SUBROUTINE_BLOCK ValveA_Diag:SBR16
TITLE=// ============================================================
// // 文件: FC30_ValveA_Diag.stl
// // 功能: 阀A诊断（差值法计量+延时验证4项并行+漫溢保护）
// // Story: AQEX-7 阀门诊断
// // 调用方: FC11(S1上缸进水)
// // 说明: 阀A不使用四态诊断，采用差值法+延时验证
// //       诊断子状态VW260: 0空闲/1等开到位/2开启完成/3运行中/5关闭后验证
// //
// // 修复记录:
// //   P1 - MOVR/-R 替换 MOVD/-D: 流量计数据为REAL浮点,之前用双整数指令导致VD90=NAN
// //   P2 - 单NETWORK合并: 所有JMP/LBL在同一NETWORK内,解决STEP7导入跨NETWORK跳转失效
// //   P3 - I8.0 去掉EU: 子状态1→2改用常开触点,PLC冷启动时阀已开到位也能正常进入子状态2
// //   P4 - 关阀快照MOVD改MOVR: 语义一致,REAL数据用MOVR搬运
// // ============================================================
// 
// // 符号说明:
// // VW260 : Diag_State_A     阀A诊断子状态
// // VW266 : Diag_Result_A    阀A诊断结果(0进行中/1正常/2故障)
// // VD308 : VD_FlowMeter_CloseSnapshot  阀A关阀瞬间流量计快照
// // VD312 : VD_FlowMeter_CloseDelta     阀A关阀后流量计差值
// // VD316 : 目标进水量(HMI设定)
// // T50   : 阀A开到位超时(100ms时基)
// // T51   : 阀A关阀后延时验证(100ms时基)
// // T52   : 开到位但无流2s确认(100ms时基)
// // I0.0  : 流量开关A(有流=ON)
// // I0.5  : 液位计A高位(漫溢=ON)
// // I8.0  : 阀A开到位反馈
// // I8.1  : 阀A关到位反馈
// // Q0.2  : 阀A(电动球阀)
// // Q0.5  : NC球阀-上缸
BEGIN
Network 1
//  ============================================================
//  NETWORK 1 - 单NETWORK版 FC30
//  所有JMP/LBL在同一NETWORK内,避免STEP7导入后跳转失效
//  ============================================================
//  ========== 第一部分: 漫溢保护(优先级最高,全程监控) ==========
LD     CPU_输入5:I0.5          // 液位计A高位=漫溢
S      V300.0, 1             // M_Alarm_Overflow_AHigh
S      V300.2, 1             // M_Alarm_NCValve_Top
R      CPU_输出5:Q0.5, 1       // 关NC球阀(切断水流)
R      CPU_输出2:Q0.2, 1       // 关阀A
MOVW   99, VW2               // 转S_ERROR
MOVB   2, VB266              // Diag_Result_A=2故障
JMP    1                     // 跳到结束
// ========== 第二部分: 子状态调度(根据VB260分发) ========== // ========== 第二部分: 子状态调度(根据VB260分发) ==========
// ★关键修复: 子状态只存在VB260中,FC11用MOVB写VB260,VB261=0 // ★关键修复: 子状态只存在VB260中,FC11用MOVB写VB260,VB261=0
//   因此VW260实际=VB260×256(如VB260=2则VW260=512),必须用LDB=字节比较 //   因此VW260实际=VB260×256(如VB260=2则VW260=512),必须用LDB=字节比较
LDB=   VB260, 0
LDB=   VB260, 0              // 子状态0: 空闲
LDB=   VB260, 1
JMP    2                     // 子状态1: 等开到位
LDB=   VB260, 2
LDB=   VB260, 1              // 子状态2: 等流量开关
LDB=   VB260, 3
JMP    3                     // 子状态3: ★运行中算VD90★
LDB=   VB260, 5
LDB=   VB260, 2              // 子状态5: 关阀后延时验证
JMP    4                     // 兜底: 非法状态跳到结束
// ========== 第三部分: 子状态0 - 空闲 ========== // ========== 第三部分: 子状态0 - 空闲 ==========
LBL    2
// 等待FC11触发置VW260=1, 无额外动作   // 等待FC11触发置VW260=1, 无额外动作
JMP    1
// ========== 第四部分: 子状态1 - 等待开到位 ========== // ========== 第四部分: 子状态1 - 等待开到位 ==========
LBL    3
// T50超时计时(PT=VW278, 由FC11计算VD358×10写入) // T50超时计时(PT=VW278, 由FC11计算VD358×10写入)
LD     SM0.0
TON    T50, VW278
// I8.0开到位反馈=ON → 转子状态2      // I8.0开到位反馈=ON → 转子状态2
// ★P3修复: 去掉EU(上升沿),改用常开触点   // ★P3修复: 去掉EU(上升沿),改用常开触点
//   正常: 阀A打开后I8.0从OFF→ON,直接触发 //   正常: 阀A打开后I8.0从OFF→ON,直接触发
//   异常: PLC冷启动时阀已开到位(I8.0本来就是ON),也能立即进入子状态2 //   异常: PLC冷启动时阀已开到位(I8.0本来就是ON),也能立即进入子状态2
LD     I8.0
LDB=   VB260, 3              // VW260=2
JMP    5                     // 清子状态索引
LDB=   VB260, 5              // 复位超时计时
JMP    1
// T50超时 → 开到位超时报警           // T50超时 → 开到位超时报警
LD     T50
JMP    6                     // M_Alarm_ValveA_OpenTimeout
MOVW   99, VW2
MOVB   2, VB266
JMP    1
// ========== 第五部分: 子状态2 - 等待流量开关 ========== // ========== 第五部分: 子状态2 - 等待流量开关 ==========
LBL    4
// I0.0流量开关A=ON → 正常有流, 转子状态3运行中 // I0.0流量开关A=ON → 正常有流, 转子状态3运行中
LD     I0.0
JMP    1                     // VW260=3运行中
MOVB   0, VB261
JMP    1
// 开到位但无流 → 加2s延时确认避免瞬时波动    // 开到位但无流 → 加2s延时确认避免瞬时波动
LBL    2                     // 阀确实已开到位
JMP    1                     // 但无流量
LBL    3                     // 2s确认(20×100ms)
LD     T52
LD     Always_On:SM0.0       // M_Alarm_ValveA_OpenNoFlow
MOVW   99, VW2
MOVB   2, VB266
JMP    1
// ========== 第六部分: 子状态3 - ★运行中差值法持续计量★ ========== // ========== 第六部分: 子状态3 - ★运行中差值法持续计量★ ==========
LBL    5
// ★P1修复: 用MOVR/-R实数指令计算进水量(原MOVD/-D导致NAN) // ★P1修复: 用MOVR/-R实数指令计算进水量(原MOVD/-D导致NAN)
// VD_Current_InletVolume(VD90) = VD86(当前累计) - VD82(开启快照) // VD_Current_InletVolume(VD90) = VD86(当前累计) - VD82(开启快照)
LD     SM0.0
TON    T50, VW278            // ★MOVR: 实数搬运
LD     EM0_输入0:I8.0          // ★-R: 实数减法
MOVB   2, VB260              // 当前进水量
// 进水量达标 → 关阀A + 快照关阀瞬间流量计值 + 转子状态5 // 进水量达标 → 关阀A + 快照关阀瞬间流量计值 + 转子状态5
LD     SM0.0
LPS
MOVB   0, VB261              // 当前进水量 ≥ 目标进水量
R      T50, 1                // 关阀A
// ★P4修复: 关阀快照也用MOVR(原MOVD虽能跑但语义不一致) // ★P4修复: 关阀快照也用MOVR(原MOVD虽能跑但语义不一致)
JMP    1                     // VD_FlowMeter_CloseSnapshot
LD     T50                   // VW260=5(关闭后验证)
MOVB   0, VB261
S      V301.4, 1             // 复位开到位无流确认计时
LPP
JMP    1
// ========== 第七部分: 子状态5 - 关阀后延时验证(4项并行) ========== // ========== 第七部分: 子状态5 - 关阀后延时验证(4项并行) ==========
LBL    6
// T51延时验证计时(PT=VW280, 由FC11计算VD66×10写入) // T51延时验证计时(PT=VW280, 由FC11计算VD66×10写入)
LD     SM0.0
TON    T51, VW280
// ★P1修复: 关阀后内漏检测也用MOVR/-R实数指令 // ★P1修复: 关阀后内漏检测也用MOVR/-R实数指令
// 持续计算关阀后流量计差值 = VD86(当前) - VD308(关阀快照) // 持续计算关阀后流量计差值 = VD86(当前) - VD308(关阀快照)
LD     SM0.0
MOVR   VD86, AC0
-R     VD308, AC0
MOVW   99, VW2               // VD_FlowMeter_CloseDelta
// --- 延时到达后4项并行校验 ---       // --- 延时到达后4项并行校验 ---
MOVB   2, VB266              // 仅T51到达时执行
LPS
// 校验1: 关阀后仍有流(流量开关A=ON)     // 校验1: 关阀后仍有流(流量开关A=ON)
A      I0.0
JMP    1                     // M_Alarm_ValveA_CloseFlow
// 校验2: 内漏(流量计差值>0.1L, 说明仍在缓慢注水) // 校验2: 内漏(流量计差值>0.1L, 说明仍在缓慢注水)
LPS
LBL    4                     // 阈值0.1L=100ml, 现场整定
LD     CPU_输入0:I0.0          // M_Alarm_ValveA_Leak
LPP
// 校验3: 关到位反馈超时(I8.1=OFF)    // 校验3: 关到位反馈超时(I8.1=OFF)
AN     I8.1
MOVB   3, VB260              // M_Alarm_ValveA_CloseTimeout
// 校验4: 关到位但仍有流(交叉验证)        // 校验4: 关到位但仍有流(交叉验证)
MOVB   0, VB261              // 阀确实关到位
JMP    1                     // 但流量开关仍有流
LD     EM0_输入0:I8.0          // M_Alarm_ValveA_CloseLeak
LPP
// --- 校验结果判定 ---            // --- 校验结果判定 ---
AN     CPU_输入0:I0.0          // T51已到
LPS
// 4项全通过: 流量开关OFF AND 差值不增 AND 关到位ON // 4项全通过: 流量开关OFF AND 差值不增 AND 关到位ON
TON    T52, 20               // 流量开关A=OFF
LD     T52                   // 差值≤0.1L(不增长=无内漏)
S      V301.5, 1             // 关到位=ON
// → 诊断正常完成                  // → 诊断正常完成
MOVW   99, VW2               // VW260=0空闲(等待下轮)
MOVB   0, VB261
MOVB   2, VB266              // Diag_Result_A=1正常完成
JMP    1                     // 复位延时计时
JMP    1
LPP
// 任一项报警 → 转S_ERROR          // 任一项报警 → 转S_ERROR
LD     T51
LBL    5                     // 4个报警标志任一为1
O      V301.1
O      V301.2
O      V301.3
LD     Always_On:SM0.0       // 转S_ERROR
MOVR   VD86, AC0             // 故障
JMP    1
// ========== 结束 ==========  // ========== 结束 ==========
LBL    1
// ============================================================ // ============================================================
// 文件结束                      // 文件结束
// 说明:                       // 说明:
//   1. FC11调用本FC前需置VW260=1启动诊断 //   1. FC11调用本FC前需置VW260=1启动诊断
//   2. FC11检查VW266: 0=进行中等待, 1=正常完成转S2, 2=故障(已转S_ERROR) //   2. FC11检查VW266: 0=进行中等待, 1=正常完成转S2, 2=故障(已转S_ERROR)
//   3. VD316(目标进水量)由HMI设定或FC11计算写入 //   3. VD316(目标进水量)由HMI设定或FC11计算写入
//   4. VW278=T50×10(开到位超时), VW280=T51×10(延时验证), 由FC11计算写入 //   4. VW278=T50×10(开到位超时), VW280=T51×10(延时验证), 由FC11计算写入
//   5. 内漏阈值0.1L为初值, 需现场整定   //   5. 内漏阈值0.1L为初值, 需现场整定
//   6. 所有JMP/LBL在单NETWORK内, 避免STEP7导入后跳转失效(P2修复) //   6. 所有JMP/LBL在单NETWORK内, 避免STEP7导入后跳转失效(P2修复)
// ============================================================

 // ============================================================
-R     VD82, AC0
MOVR   AC0, VD90
LD     Always_On:SM0.0
LPS
AR>=   VD90, VD316
R      CPU_输出2:Q0.2, 1
MOVR   VD86, VD308
MOVB   5, VB260
MOVB   0, VB261
R      T52, 1
LPP
JMP    1
LBL    6
LD     Always_On:SM0.0
TON    T51, VW280
LD     Always_On:SM0.0
MOVR   VD86, AC0
-R     VD308, AC0
MOVR   AC0, VD312
LD     T51
LPS
A      CPU_输入0:I0.0
S      V301.0, 1
LPS
AR>    VD312, 0.1
S      V301.1, 1
LPP
AN     EM0_输入1:I8.1
S      V301.2, 1
A      EM0_输入1:I8.1
A      CPU_输入0:I0.0
S      V301.3, 1
LPP
LD     T51
LPS
AN     CPU_输入0:I0.0
AR<=   VD312, 0.1
A      EM0_输入1:I8.1
MOVB   0, VB260
MOVB   0, VB261
MOVB   1, VB266
R      T51, 1
JMP    1
LPP
LD     T51
A      V301.0
O      V301.1
O      V301.2
O      V301.3
MOVW   99, VW2
MOVB   2, VB266
JMP    1
LBL    1
END_SUBROUTINE_BLOCK

SUBROUTINE_BLOCK ValveB_Diag:SBR17
TITLE=// ============================================================
// // 文件: FC31_ValveB_Diag.stl
// // 功能: 阀B诊断（四态诊断+开关到位+超时保护+漫溢保护）
// // Story: AQEX-7 阀门诊断
// // 调用方: FC15(S4上→下转移)
// // 说明: 阀B四态诊断(流量开关B+液位计A低位)
// //       诊断子状态VW262: 0空闲/1等开到位/2开启完成/3运行中/4等关到位
// // ============================================================
// 
// // 符号说明:
// // VW262 : Diag_State_B     阀B诊断子状态
// // VW268 : Diag_Result_B    阀B诊断结果(0/1/2)
// // T53   : 阀B开到位超时
// // T54   : 阀B流量开关超时保护
// // T55   : 阀B关到位超时
// // I0.1  : 流量开关B
// // I0.6  : 液位计A低位(上缸排空)
// // I0.7  : 液位计B高位(下缸漫溢)
// // I8.2  : 阀B开到位反馈
// // I8.3  : 阀B关到位反馈
// // Q0.3  : 阀B
// // Q0.6  : NC球阀-下缸
// 
BEGIN
Network 1
//  漫溢保护（全程，优先级最高）
//  液位计B高位=ON立即报警+关NC阀+关阀B+转S_ERROR
//  NC球阀与电动球阀串联冗余:高位时关闭NC球阀切断水流,防止球阀关不严持续注水
LD     CPU_输入7:I0.7
S      V300.1, 1             // M_Alarm_Overflow_BHigh
S      V300.3, 1             // M_Alarm_NCValve_Bottom(NC球阀下缸关闭报警,漫溢风险级)
R      CPU_输出6:Q0.6, 1       // 关闭下缸NC球阀(切断水流)
R      CPU_输出3:Q0.3, 1       // 关阀B
MOVW   99, VW2
MOVB   2, VB268              // 故障
JMP    1




Network 2
//  诊断子状态调度
LDW=   VW262, 0
JMP    2
LDW=   VW262, 1
JMP    3
LDW=   VW262, 2
JMP    4
LDW=   VW262, 3
JMP    5
LDW=   VW262, 4
JMP    6
JMP    1




// ---- 子状态0: 空闲 ----
       // ---- 子状态0: 空闲 ----
Network 3
//  S0空闲
LBL    2
JMP    1




// ---- 子状态1: 等待开到位 ----
    // ---- 子状态1: 等待开到位 ----
Network 4
//  S1等待开到位
LBL    3
// T53开到位超时 + T54流量开关超时(两套独立判据)
 // T53开到位超时 + T54流量开关超时(两套独立判据)
LD     Always_On:SM0.0
TON    T53, VW274            // PT=VD_Timeout_ValveB(VD362)×10
TON    T54, VW274            // 流量开关超时(同参数，独立计时)


// 开到位=ON → 转S2
             // 开到位=ON → 转S2
LD     EM0_输入2:I8.2
EU
MOVB   2, VB262
MOVB   0, VB263
R      T53, 1
R      T54, 1
JMP    1


// 开到位超时 → 报警
               // 开到位超时 → 报警
LD     T53
S      V302.1, 1             // M_Alarm_ValveB_OpenTimeout
MOVW   99, VW2
MOVB   2, VB268
JMP    1


// 流量开关超时(开阀后一直无流) → 报警
     // 流量开关超时(开阀后一直无流) → 报警
LD     T54
AN     CPU_输入1:I0.1          // 确认流量开关B仍OFF
S      V302.2, 1             // M_Alarm_ValveB_OpenNoFlow
MOVW   99, VW2
MOVB   2, VB268
JMP    1




// ---- 子状态2: 开启完成检查 ----
   // ---- 子状态2: 开启完成检查 ----
Network 5
//  S2开启完成检查
LBL    4
// 流量开关B=ON → 正常，转S3
        // 流量开关B=ON → 正常，转S3
LD     CPU_输入1:I0.1
MOVB   3, VB262
MOVB   0, VB263
JMP    1


// 开到位但无流 → 报警
              // 开到位但无流 → 报警
LD     EM0_输入2:I8.2
AN     CPU_输入1:I0.1
S      V302.2, 1             // M_Alarm_ValveB_OpenNoFlow
MOVW   99, VW2
MOVB   2, VB268
JMP    1




// ---- 子状态3: 运行中(四态诊断持续扫描) ----
 // ---- 子状态3: 运行中(四态诊断持续扫描) ----
Network 6
//  S3四态诊断
LBL    5
// 四态诊断: 流量开关B(I0.1) + 液位计A低位(I0.6)
 // 四态诊断: 流量开关B(I0.1) + 液位计A低位(I0.6)
// 状态3: 流量开关OFF + 液位低位ON → 上缸排空，关阀触发
 // 状态3: 流量开关OFF + 液位低位ON → 上缸排空，关阀触发
LD     CPU_输入6:I0.6          // 液位计A低位=ON(上缸空)
AN     CPU_输入1:I0.1          // 且流量开关B=OFF(转移结束)
R      CPU_输出3:Q0.3, 1       // 关阀B
MOVB   4, VB262              // 转S4等关到位
MOVB   0, VB263
JMP    1


// 状态4: 流量开关OFF + 液位低位OFF → 设备故障
 // 状态4: 流量开关OFF + 液位低位OFF → 设备故障
LD     CPU_输入1:I0.1          // 流量开关B
NOT
AN     CPU_输入6:I0.6          // 且液位低位OFF
// 注:需排除刚开始转移时的瞬时(流量开关尚未ON)
 // 注:需排除刚开始转移时的瞬时(流量开关尚未ON)
// 简化: 直接判定状态4
              // 简化: 直接判定状态4
S      V302.0, 1             // M_Alarm_ValveB_Diag
MOVW   99, VW2
MOVB   2, VB268
JMP    1


// 状态1/2: 流量开关ON → 正常转移中/即将排空，继续
 // 状态1/2: 流量开关ON → 正常转移中/即将排空，继续
LD     CPU_输入1:I0.1
JMP    1




// ---- 子状态4: 等待关到位 ----
    // ---- 子状态4: 等待关到位 ----
Network 7
//  S4等待关到位
LBL    6
// T55关到位超时
                 // T55关到位超时
LD     Always_On:SM0.0
TON    T55, VW274            // PT=VD_Timeout_ValveB×10


// 关到位=ON AND 流量开关=OFF → 正常完成
 // 关到位=ON AND 流量开关=OFF → 正常完成
LD     EM0_输入3:I8.3
AN     CPU_输入1:I0.1
MOVB   0, VB262              // VW262=0空闲
MOVB   0, VB263
MOVB   1, VB268              // Diag_Result_B=1正常完成
R      T55, 1
JMP    1


// 关到位=ON AND 流量开关=ON → 内漏
  // 关到位=ON AND 流量开关=ON → 内漏
LD     EM0_输入3:I8.3
A      CPU_输入1:I0.1
S      V302.4, 1             // M_Alarm_ValveB_CloseLeak
MOVW   99, VW2
MOVB   2, VB268
JMP    1


// 关到位超时 → 报警
               // 关到位超时 → 报警
LD     T55
AN     EM0_输入3:I8.3
S      V302.3, 1             // M_Alarm_ValveB_CloseTimeout
MOVW   99, VW2
MOVB   2, VB268
JMP    1




Network 8
//  诊断结束
LBL    1




// ============================================================
 // ============================================================
// 文件结束
                     // 文件结束
// 说明:
                      // 说明:
//   1. FC15调用本FC前置VW262=1启动
 //   1. FC15调用本FC前置VW262=1启动
//   2. FC15检查VW268: 0等待, 1正常完成转S5, 2故障
 //   2. FC15检查VW268: 0等待, 1正常完成转S5, 2故障
//   3. VW274=VD_Timeout_ValveB(VD362)×10转换值
 //   3. VW274=VD_Timeout_ValveB(VD362)×10转换值
//   4. 四态诊断状态4需排除转移初期瞬时，实际需加延时确认
 //   4. 四态诊断状态4需排除转移初期瞬时，实际需加延时确认
// ============================================================
 // ============================================================


END_SUBROUTINE_BLOCK

SUBROUTINE_BLOCK ValveC_Diag:SBR18
TITLE=// ============================================================
// // 文件: FC32_ValveC_Diag.stl
// // 功能: 阀C诊断（四态诊断+开关到位+超时保护）
// // Story: AQEX-7 阀门诊断
// // 调用方: FC17(S6下缸排水)
// // 说明: 阀C四态诊断(流量开关C+液位计B低位)，与阀B对称
// //       阀C无漫溢保护(下缸排水不会漫溢)
// //       诊断子状态VW264: 0空闲/1等开到位/2开启完成/3运行中/4等关到位
// // ============================================================
// 
// // 符号说明:
// // VW264 : Diag_State_C     阀C诊断子状态
// // VW270 : Diag_Result_C    阀C诊断结果(0/1/2)
// // T56   : 阀C开到位超时
// // T57   : 阀C流量开关超时保护
// // T58   : 阀C关到位超时
// // I0.2  : 流量开关C
// // I1.0  : 液位计B低位(下缸排空)
// // I8.4  : 阀C开到位反馈
// // I8.5  : 阀C关到位反馈
// // Q0.4  : 阀C
BEGIN
Network 1
//  诊断子状态调度
//  注: 阀C无漫溢保护，直接进入状态调度
LDW=   VW264, 0
JMP    1
LDW=   VW264, 1
JMP    2
LDW=   VW264, 2
JMP    3
LDW=   VW264, 3
JMP    4
LDW=   VW264, 4
JMP    5
JMP    6




// ---- 子状态0: 空闲 ----
       // ---- 子状态0: 空闲 ----
Network 2
//  S0空闲
LBL    1
JMP    6




// ---- 子状态1: 等待开到位 ----
    // ---- 子状态1: 等待开到位 ----
Network 3
//  S1等待开到位
LBL    2
// T56开到位超时 + T57流量开关超时(两套独立判据)
 // T56开到位超时 + T57流量开关超时(两套独立判据)
LD     Always_On:SM0.0
TON    T56, VW276            // PT=VD_Timeout_ValveC(VD54)×10
TON    T57, VW276            // 流量开关超时


// 开到位=ON → 转S2
             // 开到位=ON → 转S2
LD     EM0_输入4:I8.4
EU
MOVB   2, VB264
MOVB   0, VB265
R      T56, 1
R      T57, 1
JMP    6


// 开到位超时 → 报警
               // 开到位超时 → 报警
LD     T56
S      V302.6, 1             // M_Alarm_ValveC_OpenTimeout
MOVW   99, VW2
MOVW   2, VW270
JMP    6


// 流量开关超时 → 报警
              // 流量开关超时 → 报警
LD     T57
AN     CPU_输入2:I0.2
S      V302.7, 1             // M_Alarm_ValveC_OpenNoFlow
MOVW   99, VW2
MOVW   2, VW270
JMP    6




// ---- 子状态2: 开启完成检查 ----
   // ---- 子状态2: 开启完成检查 ----
Network 4
//  S2开启完成检查
LBL    3
// 流量开关C=ON → 正常，转S3
        // 流量开关C=ON → 正常，转S3
LD     CPU_输入2:I0.2
MOVB   3, VB264
MOVB   0, VB265
JMP    6


// 开到位但无流 → 报警
              // 开到位但无流 → 报警
LD     EM0_输入4:I8.4
AN     CPU_输入2:I0.2
S      V302.7, 1             // M_Alarm_ValveC_OpenNoFlow
MOVW   99, VW2
MOVW   2, VW270
JMP    6




// ---- 子状态3: 运行中(四态诊断持续扫描) ----
 // ---- 子状态3: 运行中(四态诊断持续扫描) ----
Network 5
//  S3四态诊断
LBL    4
// 四态诊断: 流量开关C(I0.2) + 液位计B低位(I1.0)
 // 四态诊断: 流量开关C(I0.2) + 液位计B低位(I1.0)
// 状态3: 流量开关OFF + 液位低位ON → 下缸排空，关阀触发
 // 状态3: 流量开关OFF + 液位低位ON → 下缸排空，关阀触发
LD     CPU_输入8:I1.0          // 液位计B低位=ON(下缸空)
AN     CPU_输入2:I0.2          // 且流量开关C=OFF(排水结束)
R      CPU_输出4:Q0.4, 1       // 关阀C
MOVB   4, VB264              // 转S4等关到位
MOVB   0, VB265
JMP    6


// 状态4: 流量开关OFF + 液位低位OFF → 设备故障
 // 状态4: 流量开关OFF + 液位低位OFF → 设备故障
LD     CPU_输入2:I0.2
NOT
AN     CPU_输入8:I1.0
S      V302.5, 1             // M_Alarm_ValveC_Diag
MOVW   99, VW2
MOVW   2, VW270
JMP    6


// 状态1/2: 流量开关ON → 正常排水中，继续
 // 状态1/2: 流量开关ON → 正常排水中，继续
LD     CPU_输入2:I0.2
JMP    6




// ---- 子状态4: 等待关到位 ----
    // ---- 子状态4: 等待关到位 ----
Network 6
//  S4等待关到位
LBL    5
// T58关到位超时
                 // T58关到位超时
LD     Always_On:SM0.0
TON    T58, VW276            // PT=VD_Timeout_ValveC×10


// 关到位=ON AND 流量开关=OFF → 正常完成
 // 关到位=ON AND 流量开关=OFF → 正常完成
LD     EM0_输入5:I8.5
AN     CPU_输入2:I0.2
MOVB   0, VB264              // VW264=0空闲
MOVB   0, VB265
MOVW   1, VW270              // Diag_Result_C=1正常完成(已修正:用MOVW写完整WORD)
R      T58, 1
JMP    6


// 关到位=ON AND 流量开关=ON → 内漏
  // 关到位=ON AND 流量开关=ON → 内漏
LD     EM0_输入5:I8.5
A      CPU_输入2:I0.2
S      V303.1, 1             // M_Alarm_ValveC_CloseLeak
MOVW   99, VW2
MOVW   2, VW270
JMP    6


// 关到位超时 → 报警
               // 关到位超时 → 报警
LD     T58
AN     EM0_输入5:I8.5
S      V303.0, 1             // M_Alarm_ValveC_CloseTimeout
MOVW   99, VW2
MOVW   2, VW270              // Diag_Result_C=2故障(已修正:用MOVW)
JMP    6




Network 7
//  诊断结束
LBL    6




// ============================================================
 // ============================================================
// 文件结束
                     // 文件结束
// 说明:
                      // 说明:
//   1. FC17调用本FC前置VW264=1启动
 //   1. FC17调用本FC前置VW264=1启动
//   2. FC17检查VW270: 0等待, 1正常完成转S5/S7, 2故障
 //   2. FC17检查VW270: 0等待, 1正常完成转S5/S7, 2故障
//   3. VW276=VD_Timeout_ValveC(VD54)×10转换值
 //   3. VW276=VD_Timeout_ValveC(VD54)×10转换值
//   4. 阀C无漫溢保护(下缸排水不漫溢)
    //   4. 阀C无漫溢保护(下缸排水不漫溢)
//   5. VW270写入统一用MOVW(写完整WORD),确保FC17的AW=VW270判断正确
 //   5. VW270写入统一用MOVW(写完整WORD),确保FC17的AW=VW270判断正确
// ============================================================
 // ============================================================


END_SUBROUTINE_BLOCK

SUBROUTINE_BLOCK RhythmCorrection:SBR19
TITLE=// ============================================================
// // 文件: FC40_RhythmCorrection.stl
// // 功能: 配液节奏三层纠偏核心算法
// // Story: AQEX-8 节奏纠偏 (AQEX-6 状态机骨架预留接口填充)
// // 说明: 纯数学算法,输入Available/Needed,输出S2/RestTime/CycleExtend目标+报警
// //       模式VW182: 0=预规划(S5上升沿触发), 1=二次校正(S1完成触发)
// //       三层额度: 第0层压缩静止等候→第1层压缩S2→第2层顺延周期
// // ============================================================
// 
// // 符号说明:
// // VW182 : VW_Corr_Mode       纠偏模式(0预规划/1二次校正)
// // VD150 : VD_Available       剩余可用时间(s) [调用方填入]
// // VD154 : VD_Needed          所需时间(s) [调用方填入]
// // VD158 : VD_Delta           缺口 = Needed - Available(s)
// // VD162 : VD_Layer0_Quota    第0层额度(静止等候可压缩量)
// // VD166 : VD_Layer1_Quota    第1层额MBUS_CTRL度(S2可压缩量)
// // VD170 : VD_Layer2_Quota    第2层额度(周期可顺延量,s)
// // VD120 : VD_S2_Target       输出:本轮S2目标时长(s)
// // VD124 : VD_RestTime_Target 输出:本轮S3.5目标时长(s)
// // VD128 : VD_CycleExtend_Target 输出:允许下缸空等时长(min)
// // VW184 : VW_Corr_Result     输出:0进行中/1正常/2已纠偏/3滞后提示/4人工介入
// // V300.6: M_Alarm_ScheduleLag     严重滞后(人工介入)报警
// // V300.7: M_Alarm_ScheduleLag_Warn 滞后提示报警
// 
BEGIN
Network 1
//  计算三层额度 + 清结果
LD     Always_On:SM0.0
MOVW   0, VW184              // 清纠偏结果
// 第0层额度 = VD_RestTime - VD_RestTime_Min
 // 第0层额度 = VD_RestTime - VD_RestTime_Min
MOVR   VD36, VD162           // VD_RestTime
-R     VD40, VD162           // - VD_RestTime_Min
// 第1层额度 = VD_PreMixTime - VD_PreMixTime_MinSafe
 // 第1层额度 = VD_PreMixTime - VD_PreMixTime_MinSafe
MOVR   VD28, VD166           // VD_PreMixTime
-R     VD32, VD166           // - VD_PreMixTime_MinSafe
// 第2层额度 = VD_CycleExtend_Max × 60 (min→s)
 // 第2层额度 = VD_CycleExtend_Max × 60 (min→s)
MOVR   VD44, VD170           // VD_CycleExtend_Max(min)
*R     60.0, VD170           // →秒




Network 2
//  判断是否需要纠偏(Available >= Needed → 无需纠偏)
LD     Always_On:SM0.0
AR>=   VD150, VD154          // Available >= Needed ?
JMP    1                     // 是 → 无需纠偏
// 否 → 继续计算缺口
               // 否 → 继续计算缺口




Network 3
//  计算缺口Delta + 第0层扣减(压缩静止等候)
LD     Always_On:SM0.0
// Delta = Needed - Available
 // Delta = Needed - Available
MOVR   VD154, VD158          // Delta = Needed
-R     VD150, VD158          // - Available
// 第0层判断: Delta <= Layer0_Quota ?
 // 第0层判断: Delta <= Layer0_Quota ?
LD     Always_On:SM0.0
AR<=   VD158, VD162          // Delta <= 第0层额度 ?
JMP    2                     // 是 → 第0层够
// 否 → 第0层用满,Delta减去第0层额度,继续第1层
 // 否 → 第0层用满,Delta减去第0层额度,继续第1层
LD     Always_On:SM0.0
MOVR   VD40, VD124           // VD_RestTime_Target = VD_RestTime_Min(用满)
MOVR   VD158, AC0            // 暂存Delta
-R     VD162, AC0            // Delta - Layer0_Quota
MOVR   AC0, VD158            // 更新Delta
JMP    3                     // → 第1层


LBL    2
LD     Always_On:SM0.0
MOVR   VD36, VD124           // VD_RestTime_Target = VD_RestTime - Delta
-R     VD158, VD124
MOVR   VD28, VD120           // VD_S2_Target = VD_PreMixTime(不动)
MOVR   0.0, VD128            // VD_CycleExtend_Target = 0
MOVB   2, VB184              // Result=2(已纠偏)
JMP    4




Network 4
//  第1层扣减(压缩S2预循环)
LBL    3
LD     Always_On:SM0.0
AR<=   VD158, VD166          // Delta <= 第1层额度 ?
JMP    5                     // 是 → 第1层够
// 否 → 第1层用满,Delta减去第1层额度,继续第2层
 // 否 → 第1层用满,Delta减去第1层额度,继续第2层
LD     Always_On:SM0.0
MOVR   VD32, VD120           // VD_S2_Target = VD_PreMixTime_MinSafe(用满)
MOVR   VD158, AC0            // 暂存Delta
-R     VD166, AC0            // Delta - Layer1_Quota
MOVR   AC0, VD158            // 更新Delta
JMP    6                     // → 第2层


LBL    5
LD     Always_On:SM0.0
MOVR   VD28, VD120           // VD_S2_Target = VD_PreMixTime - Delta
-R     VD158, VD120
MOVR   0.0, VD128            // VD_CycleExtend_Target = 0
MOVB   2, VB184              // Result=2(已纠偏)
JMP    4




Network 5
//  第2层扣减(顺延换水周期)
LBL    6
LD     Always_On:SM0.0
AR<=   VD158, VD170          // Delta <= 第2层额度(总顺延上限) ?
JMP    7                     // 是 → 顺延可覆盖
// 否 → 三层额度全部用尽,人工介入
        // 否 → 三层额度全部用尽,人工介入
LD     Always_On:SM0.0
MOVB   4, VB184              // Result=4(人工介入)
S      V300.6, 1             // M_Alarm_ScheduleLag(严重滞后,强制人工确认)
MOVW   99, VW2               // 转S_ERROR(VW2=99)
JMP    4


LBL    7
// 顺延周期可覆盖,触发滞后提示报警
         // 顺延周期可覆盖,触发滞后提示报警
LD     Always_On:SM0.0
MOVR   VD158, VD128          // VD_CycleExtend_Target = Delta(s)
/R     60.0, VD128           // →min写回
MOVB   3, VB184              // Result=3(滞后提示)
// 滞后提示报警:预规划已置位则不重复(二次校正微调场景)
 // 滞后提示报警:预规划已置位则不重复(二次校正微调场景)
LD     Always_On:SM0.0
AN     V300.7                // 预规划未触发过滞后提示?
S      V300.7, 1             // 才置位(避免二次校正重复报警)
JMP    4




Network 6
//  无需纠偏分支(Available >= Needed)
LBL    1
LD     Always_On:SM0.0
MOVR   VD28, VD120           // VD_S2_Target = VD_PreMixTime(标称)
MOVR   VD36, VD124           // VD_RestTime_Target = VD_RestTime(标称)
MOVR   0.0, VD128            // VD_CycleExtend_Target = 0(无需顺延)
MOVB   1, VB184              // Result=1(正常无需纠偏)




Network 7
//  纠偏计算结束
LBL    4
// 返回调用方(FC16预规划 或 FC11二次校正)
 // 返回调用方(FC16预规划 或 FC11二次校正)
// 调用方检查VW184:
              // 调用方检查VW184:
//   1=正常 → 按标称执行
           //   1=正常 → 按标称执行
//   2=已纠偏 → 按Target执行
      //   2=已纠偏 → 按Target执行
//   3=滞后提示 → 按Target执行,HMI显示顺延量
 //   3=滞后提示 → 按Target执行,HMI显示顺延量
//   4=人工介入 → FC40已转S_ERROR,调用方本周期结束
 //   4=人工介入 → FC40已转S_ERROR,调用方本周期结束




// ============================================================
 // ============================================================
// 文件结束
                     // 文件结束
// 说明:
                      // 说明:
//   1. 本FC为纯数学算法,不读取RTC/不操作阀门,时间由调用方(FC16)准备
 //   1. 本FC为纯数学算法,不读取RTC/不操作阀门,时间由调用方(FC16)准备
//   2. AR>=/AR<=为A型浮点比较,前需LD压栈,JMP为条件跳转(栈顶=1跳转)
 //   2. AR>=/AR<=为A型浮点比较,前需LD压栈,JMP为条件跳转(栈顶=1跳转)
//   3. V300.6(严重滞后)由本FC置位,转S_ERROR;复位由FC3人工确认后执行
 //   3. V300.6(严重滞后)由本FC置位,转S_ERROR;复位由FC3人工确认后执行
//   4. V300.7(滞后提示)二次校正不重复置位,体现7.3"不重复触发滞后报警"
 //   4. V300.7(滞后提示)二次校正不重复置位,体现7.3"不重复触发滞后报警"
//   5. 单位:内部统一秒,VD_CycleExtend_Target输出min(÷60写回)
 //   5. 单位:内部统一秒,VD_CycleExtend_Target输出min(÷60写回)
// ============================================================
 // ============================================================


END_SUBROUTINE_BLOCK

// SBR20: protected block, not included

// SBR21: protected block, not included

// SBR22: protected block, not included

SUBROUTINE_BLOCK ManualSyringePump:SBR23
TITLE=FC21
BEGIN
Network 1
//  孤儿态自恢复
LDW<>  VW390, 0
AW<>   VW390, 30
AN     M11.6
AN     M11.7
AN     M12.0
AN     M13.5
AN     M13.6
MOVW   0, VW390
INCW   VW548
R      M13.7, 1
INCW   VW516




Network 2
//  启动命令检测 - 仅空闲态(VW390=0)响应
LD     Always_On:SM0.0
A      V307.2
EU
AW=    VW390, 0
MOVR   0.0, VD392
MOVR   VD452, VD396
R      M13.7, 1
R      M13.5, 1
R      M13.6, 1
R      M12.0, 1
R      M11.6, 1
R      M11.7, 1
MOVW   1, VW390
R      V307.2, 1
INCW   VW524




Network 3
//  停止命令检测 - 非空闲态响应
LD     Always_On:SM0.0
A      V307.3
EU
AW<>   VW390, 0
S      M13.7, 1
R      V307.3, 1
INCW   VW526




Network 4
//  全局错误检测
LDW=   VW390, 1
OW=    VW390, 2
OW=    VW390, 3
LD     V303.4
LD     Always_On:SM0.0
AW>=   VW4, 4
OLD
ALD
MOVW   99, VW390
R      M13.5, 1
R      M13.6, 1
R      M13.7, 1
R      M12.0, 1
R      M11.6, 1
R      M11.7, 1




Network 5
//  子状态1-1 - 计算本次抽液步数
LD     Always_On:SM0.0
AW=    VW390, 1
AN     M13.5
AN     M11.6
AN     M11.7
AN     M12.0
MOVR   VD396, VD102
/R     VD350, VD102
AR>=   VD102, 6000.0
JMP    10
ROUND  VD102, AC0
MOVR   AC0, VD102
JMP    11
LBL    10
MOVR   6000.0, VD102
LBL    11
INCW   VW528




Network 6
//  子状态1-2 - 检查步数并下发抽液指令(40006)
LD     Always_On:SM0.0
AW=    VW390, 1
AN     M13.5
AN     M11.6
AN     M11.7
AN     M12.0
AW=    VW4, 0
=      V60.4
LD     V60.4
ROUND  VD102, AC0
AR>    AC0, 0.0
JMP    12
LD     V60.4
R      M12.0, 1
R      M11.6, 1
R      M11.7, 1
MOVW   3, VW390
INCW   VW532
JMP    13
LBL    12
MOVW   AC0, VW204
MOVW   AC0, VW230
MOVD   16#9C46, VD232
S      M11.6, 1
S      M13.5, 1
LBL    13
INCW   VW530




Network 7
//  子状态1-3 - 抽液写失败处理
LD     M12.0
AW=    VW390, 1
A      V303.4
MOVW   99, VW390
R      M13.5, 1
R      M13.7, 1
R      M12.0, 1
R      M11.6, 1
R      M11.7, 1




Network 8
//  子状态1-3 - 抽液写成功处理
LD     M12.0
AW=    VW390, 1
AN     V303.4
R      M12.0, 1
R      M11.6, 1




Network 9
//  子状态1-4 - 等待抽液执行完成
LD     M13.5
AW=    VW390, 1
AW=    VW4, 0
AN     M11.6
AN     M11.7
AN     M12.0
R      M13.5, 1
MOVW   2, VW390
INCW   VW534




Network 10
//  子状态2-1 - 下发排液指令(40007)
LD     Always_On:SM0.0
AW=    VW390, 2
AN     M13.6
AN     M11.6
AN     M11.7
AN     M12.0
AW=    VW4, 0
ROUND  VD102, AC0
MOVW   AC0, VW230
MOVW   AC0, VW206
MOVD   16#9C47, VD232
S      M11.6, 1
S      M13.6, 1
INCW   VW536




Network 11
//  子状态2-2 - 排液写失败处理
LD     M12.0
AW=    VW390, 2
A      V303.4
MOVW   99, VW390
R      M13.6, 1
R      M13.7, 1
R      M12.0, 1
R      M11.6, 1
R      M11.7, 1




Network 12
//  子状态2-2 - 排液写成功处理
LD     M12.0
AW=    VW390, 2
AN     V303.4
R      M12.0, 1
R      M11.6, 1




Network 13
//  子状态2-3 - 等待排液执行完成,累加本循环体积
LD     M13.6
AW=    VW390, 2
AW=    VW4, 0
AN     M11.6
AN     M11.7
AN     M12.0
MOVR   VD102, AC0
*R     VD350, AC0
+R     AC0, VD392
-R     AC0, VD396
R      M13.6, 1
INCW   VW538




Network 14
//  子状态2-4 - 判断分支: 停止请求 → 回零
LD     Always_On:SM0.0
AW=    VW390, 2
AN     M13.6
A      M13.7
R      M12.0, 1
R      M11.6, 1
R      M11.7, 1
MOVW   3, VW390
INCW   VW540




Network 15
//  子状态2-4 - 判断分支: 单次模式 → 回零
LD     Always_On:SM0.0
AW=    VW390, 2
AN     M13.6
AW=    VW388, 0
R      M12.0, 1
R      M11.6, 1
R      M11.7, 1
MOVW   3, VW390
INCW   VW542




Network 16
//  子状态2-4 - 判断分支: 循环模式且累计>=目标 → 回零
LD     Always_On:SM0.0
AW=    VW390, 2
AN     M13.6
AW=    VW388, 1
AR>=   VD392, VD452
R      M12.0, 1
R      M11.6, 1
R      M11.7, 1
MOVW   3, VW390
INCW   VW544




Network 17
//  子状态2-4 - 判断分支: 循环模式且未完成 → 返回子状态1
LD     Always_On:SM0.0
AW=    VW390, 2
AN     M13.6
AW=    VW388, 1
AR<    VD392, VD452
R      M12.0, 1
R      M11.6, 1
R      M11.7, 1
MOVW   1, VW390
INCW   VW546




Network 18
//  子状态3-1 - 下发回零(复位)指令 40003=1
LD     Always_On:SM0.0
LDW=   VW390, 3
OW=    VW390, 30
AN     M11.6
AN     M11.7
AN     M12.0
AW=    VW4, 0
AW=    VW510, 0
O      T104
MOVW   1, VW230
MOVD   16#9C43, VD232
S      M11.6, 1
MOVW   30, VW390
INCW   VW518




Network 19
//  T104冷却定时器
LD     M12.0
AW=    VW390, 30
AW>    VW510, 0
TON    T104, 50




Network 20
//  子状态3-2 - 回零写失败处理
LD     M12.0
AW=    VW390, 30
A      V303.4
MOVW   99, VW390
R      M13.7, 1
R      M12.0, 1
R      M11.6, 1
R      M11.7, 1
R      T104, 1
INCW   VW522




Network 21
//  子状态3-2 - 回零写成功处理
LD     M12.0
AW=    VW390, 30
AN     V303.4
R      M12.0, 1
R      M13.5, 1
R      M13.6, 1
R      M13.7, 1
R      M11.6, 1
R      M11.7, 1
R      T104, 1
MOVW   4, VW390
INCW   VW520


END_SUBROUTINE_BLOCK

DATA_BLOCK_TAB 页面_1
BEGIN
//数据页注释
//按 F1 获取帮助和示例数据页
VD350    4.1667              // 25ml注射器单步分辨率
END_DATA_BLOCK_TAB
